Yaskawa INFORM job: TACK-2-FRONTS2-0.JBI

/JOB
//NAME TACK-2-FRONTS2-0
//POS
///NPOS 0,0,0,8,1,1
///USER 10
///TOOL 0
///POSTYPE USER
///RECTAN
///RCONF 0,0,0,0,0,0,0,0,0,0,0,0,0,0,0,0,0,0,0,0,0,0,0,0
P00049=2.600,0.000,0.000,0.0000,0.0000,0.0000
///USER 11
///RCONF 1,0,0,0,0,0,0,0,0,0,0,0,0,0,0,0,0,0,0,0,0,0,0,0
P00060=-253.149,0.000,36.500,0.0000,0.0000,90.0000
P00061=-253.150,-300.000,36.500,0.0000,15.0000,90.0000
P00062=-253.150,-100.000,36.500,0.0000,15.0000,90.0000
P00063=-255.149,0.000,29.500,0.0000,0.0000,90.0000
///POSTYPE PULSE
///PULSE
P00064=46607,-42266,-30628,-33826,21207,4644
P00065=48226,-50400,-34353,-49819,22438,75691
///USER 20
///POSTYPE USER
///RECTAN
P00066=-253.150,100.000,36.500,0.0000,15.0000,-80.0000
///POSTYPE BASE
///RCONF 0,0,0,0,0,0,0,0,0,0,0,0,0,0,0,0,0,0,0,0,0,0,0,0
BP00060=1650.000
///POSTYPE ANGLE
///ANGLE
EX00000=0.0000
//INST
///DATE 2018/11/20 18:15
///ATTR SC,RW
///GROUP1 RB1,BS1
///GROUP2 ST2
///LVARS 20,5,20,0,0,0,0,0
NOP
SFTOF
'***** tack 1
'calculate user frame
SET D015 0
CALL JOB:UF-STATION-2
'*****
'get sensor lengt
SET LD000 D011
'get weld diameter
SET LD001 D012
'*****
MUL LD000 -100
MUL LD001 100
DIV LD000 2
DIV LD001 2
ADD LD001 15000
SETE P060 (1) LD000
SETE P060 (2) 0
SETE P060 (3) LD001
SETE P060 (4) 0
SETE P060 (5) 0
SETE P060 (6) -800000
'**
SET P061 P060
SETE P061 (2) 300000
SETE P061 (5) 150000
SET P066 P061
SETE P066 (2) 550000
SETE P066 (1) -800000
'**
SETE BP060 (1) 1650000
'**
MOVL P061 BP060 V=83.3 PL=0  +MOVJ EX000
MOVL P066 BP060 V=333.3  +MOVJ EX000
MOVJ P064 BP060 VJ=15.00  +MOVJ EX000
'calculate user frame
SET D015 -1400000
CALL JOB:UF-STATION-2
SETE P061 (2) -350000
SETE P066 (2) -450000
SETE P060 (6) 850000
SETE P061 (6) 800000
SETE P066 (6) 800000
SETE P061 (5) 100000
MOVL P061 BP060 V=250.0 PL=0  +MOVJ EX000
'** correctie
GETE LD000 P060 (1)
ADD LD000 1
SETE P060 (1) LD000
SFTON P049 UF#(20)
MOVL P060 BP060 V=83.3 PL=0  +MOVJ EX000
'**
'get weld diameter
SET LD001 D012
MUL LD001 100
DIV LD001 2
'** start hoogte
ADD LD001 3000
SET P062 P060
SETE P062 (3) LD001
'**
'** welding speed
SET LI000 D013
MUL LI000 1
'** AVC value
SET LI001 D014
MUL LI001 100
GETE LD000 P062 (1)
ADD LD000 6000
SETE P062 (1) LD000
'**
MOVL P062 BP060 V=16.7 PL=0  +MOVJ EX000  //start position
MACRO1 MJ#(5) ARGF2
ARCON
AOVRON TCH#(3) TV=I001
IMOV P063 V=LI000 TF
ACOROF
ARCOF
TIMER T=3.00
MACRO1 MJ#(5) ARGF2
SETE P061 (5) 200000
'********************************
MOVL P060 BP060 V=16.7 PL=0  +MOVJ EX000
SFTOF
MOVL P061 BP060 V=83.3 PL=0  +MOVJ EX000
MOVL P066 BP060 V=83.3 PL=0  +MOVJ EX000
MOVJ P064 BP060 VJ=11.11 PL=0  +MOVJ EX000
MOVJ P065 BP060 VJ=15.00  +MOVJ EX000
'calculate user frame
SET D015 0
CALL JOB:UF-STATION-2
SETE P066 (2) 450000
SETE P061 (2) 350000
SETE P066 (6) -800000
SETE P061 (6) -800000
SETE P061 (5) 150000
MOVL P066 BP060 V=166.7 PL=0  +MOVJ EX000
MOVL P061 BP060 V=166.7 PL=0  +MOVJ EX000
END
